% RSLogix 500 project P2.RSS, saved by version 12.00.00.00 %
PROJECT "UNTITLED"    % processor: Bul.1763 MicroLogix 1100 Series B %

PROGRAM FILES
  LAD 2   3 rungs
  LAD 3 "IO"  8 rungs
  LAD 4 "CTRL"  10 rungs

DATA FILES
  O0 OUTPUT  4 elements
  I1 INPUT  6 elements
  S2 STATUS  66 elements
  B3 BINARY  1 elements
  T4 TIMER  1 elements
  C5 COUNTER  1 elements
  R6 CONTROL  1 elements
  N7 INTEGER  1 elements
  F8 FLOAT  1 elements

LADDER 2
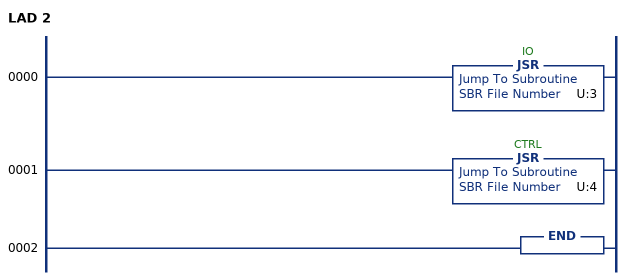
% Rung: 0 %
SOR JSR U:3 EOR
%   U:3  "IO" %
% Rung: 1 %
SOR JSR U:4 EOR
%   U:4  "CTRL" %
% Rung: 2 %
SOR END EOR

LADDER 3 "IO"
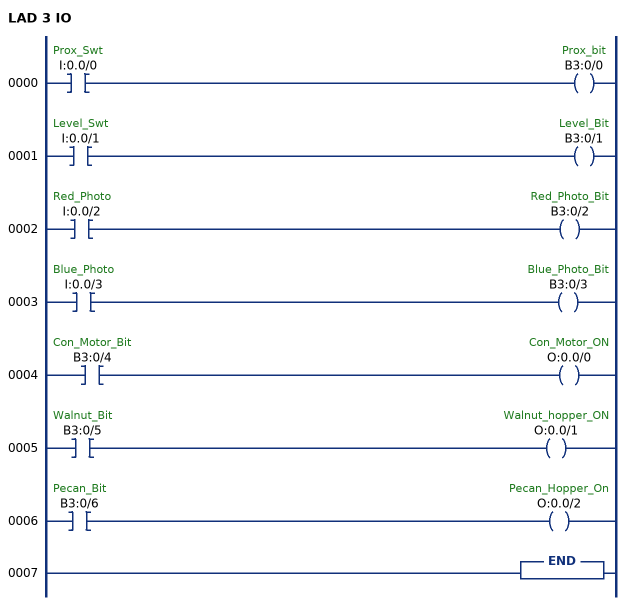
% Rung: 0 %
SOR XIC I:0.0/0 OTE B3:0/0 EOR
%   I:0.0/0  "Prox_Swt" %
%   B3:0/0  "Prox_bit" %
% Rung: 1 %
SOR XIC I:0.0/1 OTE B3:0/1 EOR
%   I:0.0/1  "Level_Swt" %
%   B3:0/1  "Level_Bit" %
% Rung: 2 %
SOR XIC I:0.0/2 OTE B3:0/2 EOR
%   I:0.0/2  "Red_Photo" %
%   B3:0/2  "Red_Photo_Bit" %
% Rung: 3 %
SOR XIC I:0.0/3 OTE B3:0/3 EOR
%   I:0.0/3  "Blue_Photo" %
%   B3:0/3  "Blue_Photo_Bit" %
% Rung: 4 %
SOR XIC B3:0/4 OTE O:0.0/0 EOR
%   B3:0/4  "Con_Motor_Bit" %
%   O:0.0/0  "Con_Motor_ON" %
% Rung: 5 %
SOR XIC B3:0/5 OTE O:0.0/1 EOR
%   B3:0/5  "Walnut_Bit" %
%   O:0.0/1  "Walnut_hopper_ON" %
% Rung: 6 %
SOR XIC B3:0/6 OTE O:0.0/2 EOR
%   B3:0/6  "Pecan_Bit" %
%   O:0.0/2  "Pecan_Hopper_On" %
% Rung: 7 %
SOR END EOR

LADDER 4 "CTRL"
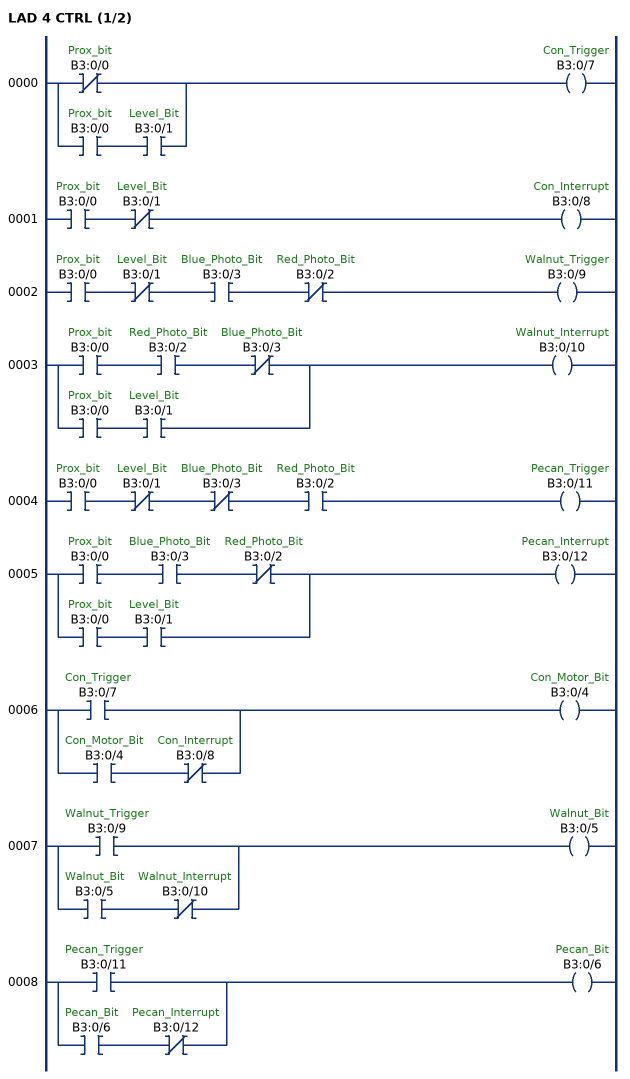
% Rung: 0 %
SOR BST XIO B3:0/0 NXB XIC B3:0/0 XIC B3:0/1 BND OTE B3:0/7 EOR
%   B3:0/0  "Prox_bit" %
%   B3:0/1  "Level_Bit" %
%   B3:0/7  "Con_Trigger" %
% Rung: 1 %
SOR XIC B3:0/0 XIO B3:0/1 OTE B3:0/8 EOR
%   B3:0/0  "Prox_bit" %
%   B3:0/1  "Level_Bit" %
%   B3:0/8  "Con_Interrupt" %
% Rung: 2 %
SOR XIC B3:0/0 XIO B3:0/1 XIC B3:0/3 XIO B3:0/2 OTE B3:0/9 EOR
%   B3:0/0  "Prox_bit" %
%   B3:0/1  "Level_Bit" %
%   B3:0/3  "Blue_Photo_Bit" %
%   B3:0/2  "Red_Photo_Bit" %
%   B3:0/9  "Walnut_Trigger" %
% Rung: 3 %
SOR BST XIC B3:0/0 XIC B3:0/2 XIO B3:0/3 NXB XIC B3:0/0 XIC B3:0/1 BND OTE B3:0/10 EOR
%   B3:0/0  "Prox_bit" %
%   B3:0/2  "Red_Photo_Bit" %
%   B3:0/3  "Blue_Photo_Bit" %
%   B3:0/1  "Level_Bit" %
%   B3:0/10  "Walnut_Interrupt" %
% Rung: 4 %
SOR XIC B3:0/0 XIO B3:0/1 XIO B3:0/3 XIC B3:0/2 OTE B3:0/11 EOR
%   B3:0/0  "Prox_bit" %
%   B3:0/1  "Level_Bit" %
%   B3:0/3  "Blue_Photo_Bit" %
%   B3:0/2  "Red_Photo_Bit" %
%   B3:0/11  "Pecan_Trigger" %
% Rung: 5 %
SOR BST XIC B3:0/0 XIC B3:0/3 XIO B3:0/2 NXB XIC B3:0/0 XIC B3:0/1 BND OTE B3:0/12 EOR
%   B3:0/0  "Prox_bit" %
%   B3:0/3  "Blue_Photo_Bit" %
%   B3:0/2  "Red_Photo_Bit" %
%   B3:0/1  "Level_Bit" %
%   B3:0/12  "Pecan_Interrupt" %
% Rung: 6 %
SOR BST XIC B3:0/7 NXB XIC B3:0/4 XIO B3:0/8 BND OTE B3:0/4 EOR
%   B3:0/7  "Con_Trigger" %
%   B3:0/4  "Con_Motor_Bit" %
%   B3:0/8  "Con_Interrupt" %
% Rung: 7 %
SOR BST XIC B3:0/9 NXB XIC B3:0/5 XIO B3:0/10 BND OTE B3:0/5 EOR
%   B3:0/9  "Walnut_Trigger" %
%   B3:0/5  "Walnut_Bit" %
%   B3:0/10  "Walnut_Interrupt" %
% Rung: 8 %
SOR BST XIC B3:0/11 NXB XIC B3:0/6 XIO B3:0/12 BND OTE B3:0/6 EOR
%   B3:0/11  "Pecan_Trigger" %
%   B3:0/6  "Pecan_Bit" %
%   B3:0/12  "Pecan_Interrupt" %

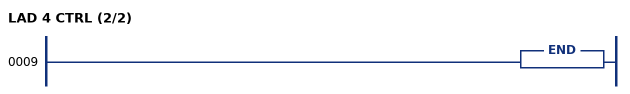
% Rung: 9 %
SOR END EOR
